FUNCTION_BLOCK FB_TOR_MS EXTENDS FB_TOR_Base
//////////////////
//  Motion Sensor System
//////////////////

VAR_INPUT PERSISTENT
	// Parameters of the Object (instance/model specific) 
		ParamTempoDoorAlarm			: TIME := T#10S ;	(* (S) Tempo for Door sensor alarm *)
		ParamTempoUnlockAlarm		: TIME := T#1800S ;	(* (S) Tempo for Door sensor alarm *)
END_VAR

VAR_OUTPUT
	//Child objects
	
END_VAR

VAR_INPUT
	// I/O Inputs 		                                     				
			MesDataExd			: TOR_Standard ;  
	
END_VAR

VAR
	//M_ALARMMANAGEMENT VARIABLES//
	
		TON_Fermeture			: TON;				//(NA) Tempo to detect door opened for too long time . 
		PT_Unlock_Alarm			: TP;				//(NA) Timer to unlock alarm after 30 min
		

END_VAR

METHOD M_AlarmManagement
//////////////////
// Manages Door sensor alarms and warnings
/////////////////

VAR 
	// Method local variables (reinitialized at each cycle) 
	FB_AlarmCodeManager : FB_AlarmCodeManager ; 

END_VAR
// Detection Variables

// The Motion Sensor must be activated for the duration of ParamTempoDoorAlarm for the alarm to be activated
TON_Fermeture(IN:= MesDataExd.MesData.MesAlarmState,PT:=ParamTempoDoorAlarm); //

// ALARM CODE //
	FB_AlarmCodeManager(
 		bAlarm1			:= FALSE,    							// 
		bAlarm2			:= FALSE, 								// 
		bAlarm3			:= FALSE, 								// 
		bAlarm4			:= FALSE, 								// 
		bAlarm5			:= FALSE,    							// 
		bAlarm6			:= FALSE, 								// 
		bAlarm7			:= FALSE, 								// 
		bAlarm8			:= FALSE, 								// 
		bAlarm9			:= FALSE,    							// 
		bAlarm10		:= FALSE, 								// 
		bAlarm11		:= FALSE, 								// 
		bAlarm12		:= FALSE, 								// 
		bAlarm13		:= FALSE,								// 
		bAlarm14		:= FALSE,								// 
		bAlarm15		:= FALSE,								// 
		wAlarmCode		=>MesDataExd.MesData.MesAlarmCode);

// WARNING CODE //
	FB_AlarmCodeManager(
		bAlarm1			:= FALSE,   							//
		bAlarm2			:= FALSE, 								// 
		bAlarm3			:= FALSE, 								// 
		bAlarm4			:= FALSE, 								// 
		bAlarm5			:= FALSE,    							// 
		bAlarm6			:= FALSE, 								// 
		bAlarm7			:= FALSE, 								// 
		bAlarm8			:= FALSE, 								// 
		bAlarm9			:= FALSE,    							// 
		bAlarm10		:= FALSE, 								// 
		bAlarm11		:= FALSE, 								// 
		bAlarm12		:= FALSE, 								// 
		bAlarm13		:= FALSE,     							//
		bAlarm14		:= FALSE,  								//
		bAlarm15		:= FALSE,  								//
		wAlarmCode		=>MesDataExd.MesData.MesWarningCode);

// EVENT CODE //
	FB_AlarmCodeManager(
		bAlarm1			:= TON_Fermeture.Q AND NOT PT_Unlock_Alarm.Q, 	// Intrusion Detected
		bAlarm2			:= FALSE, 										// 
		bAlarm3			:= FALSE, 										// 
		bAlarm4			:= FALSE, 										// 
		bAlarm5			:= FALSE,    									// 
		bAlarm6			:= FALSE, 										// 
		bAlarm7			:= FALSE, 										// 
		bAlarm8			:= FALSE, 										// 
		bAlarm9			:= FALSE,    									// 
		bAlarm10		:= FALSE, 										// 
		bAlarm11		:= FALSE, 										// 
		bAlarm12		:= FALSE, 										// 
		bAlarm13		:= FALSE,     									// 
		bAlarm14		:= FALSE,  										// 
		bAlarm15		:= FALSE,  										// 
		wAlarmCode		=>MesDataExd.MesData.MesEventCode);
		
// When the alarm is activated for the first time, it is disabled for the duration of ParamTempoUnlockAlarm to avoid spamming alarms

PT_Unlock_Alarm(IN := TON_Fermeture.Q, PT := ParamTempoUnlockAlarm);
END_METHOD

METHOD M_Execute
//////////////////
//  Method Calls 
/////////////////

VAR 
	// Method local variables (reinitialized at each cycle) 
	
END_VAR

SUPER^.M_Execute() ;
END_METHOD

METHOD M_StateManager
//////////////////
// Detect when fire occurs
/////////////////

VAR 
	// Method local variables (reinitialized at each cycle)
 	MesStateInterm1 : BOOL;
	MesStateInterm2 : BOOL;
END_VAR

IF ParamCableCutSecurity THEN
	MesStateInterm1 := NOT IN_MesState1_IO ; 
	MesStateInterm2 := NOT IN_MesState2_IO ; 
ELSE 
	MesStateInterm1 := IN_MesState1_IO;
	MesStateInterm2 := IN_MesState2_IO;
END_IF

IF ParamNbSensors = 1 THEN 
	MesStateInterm2 := MesStateInterm1 ;
END_IF

IF ParamAtleastOne THEN 
MesDataExd.MesData.MesAlarmState := MesStateInterm1 OR MesStateInterm2 ; 
ELSE
MesDataExd.MesData.MesAlarmState := MesStateInterm1 AND MesStateInterm2 ; 
END_IF

R_TRIGAlarm(CLK:= MesDataExd.MesData.MesAlarmState ) ; 
IF R_TRIGAlarm.Q THEN
	MesCountAlarm :=  MIN(MesCountAlarm + 1 ,4294967295 ) ; 
ELSIF IN_ResetCounter THEN 
	MesCountAlarm := 0 ; 
END_IF

MesDataExd.MesData.MesCountAlarm	:= MesCountAlarm ;
END_METHOD

END_FUNCTION_BLOCK

(* stored: Version 1.1.0.1, ProductVersion 3.1.4024.12
   POU FB_TOR_MS: Id {fc24f2dd-8446-4234-a094-9bc87d7f7d3c}, SpecialFunc None
   Method M_AlarmManagement: Id {88a3f6da-8e19-44f1-8279-749c28a67586}
   Method M_Execute: Id {00261c82-d7e7-4a63-8815-e22815b6b6f0}
   Method M_StateManager: Id {2a13441b-2f4a-471f-840f-f3d7c27fa4f1} *)
